INTERFACE PUBLIC MoveCommand EXTENDS AsyncCommand

{attribute 'monitoring' := 'call'}
PROPERTY PUBLIC Active : BOOL
GET
END_GET
END_PROPERTY

END_INTERFACE

(* stored: Version 1.1.0.1
   Itf MoveCommand: Id {07d8a13b-72f8-0c09-155b-77cec9d4c2ed}
   Property Active: Id {5e61e82e-e49e-0a63-19c1-b1cac31b367a}
   Get Get: Id {89635625-ce37-0a1a-2ec1-8520494e0172} *)
